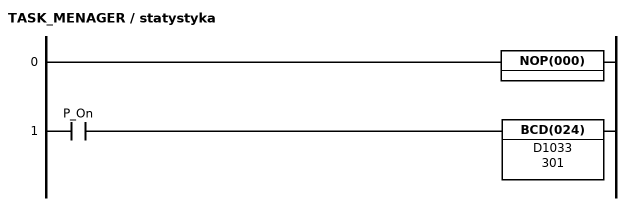
; [picture p24: TASK_MENAGER / statystyka, rungs 0-1]
; rung 0
NOP(000)
; rung 1
LD P_On
BCD(024) D1033 301

### Section wyświetlacz

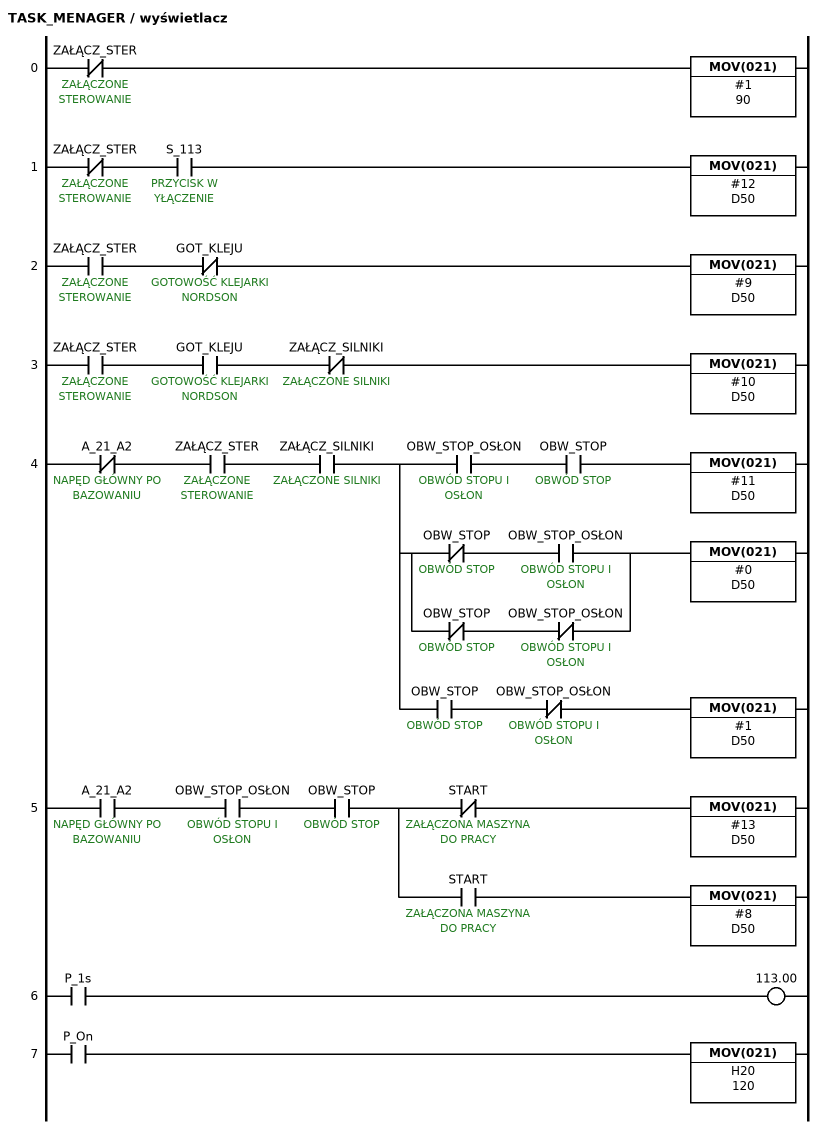
; rung 0
LDNOT ZAŁĄCZ_STER  ; ZAŁĄCZONE STEROWANIE
MOV(021) #1 90
; rung 1
LDNOT ZAŁĄCZ_STER  ; ZAŁĄCZONE STEROWANIE
AND S_113  ; PRZYCISK W YŁĄCZENIE
MOV(021) #12 D50
; rung 2
LD ZAŁĄCZ_STER  ; ZAŁĄCZONE STEROWANIE
ANDNOT GOT_KLEJU  ; GOTOWOŚĆ KLEJARKI NORDSON
MOV(021) #9 D50
; rung 3
LD ZAŁĄCZ_STER  ; ZAŁĄCZONE STEROWANIE
AND GOT_KLEJU  ; GOTOWOŚĆ KLEJARKI NORDSON
ANDNOT ZAŁĄCZ_SILNIKI  ; ZAŁĄCZONE SILNIKI
MOV(021) #10 D50
; rung 4
LDNOT A_21_A2  ; NAPĘD GŁÓWNY PO BAZOWANIU
AND ZAŁĄCZ_STER  ; ZAŁĄCZONE STEROWANIE
AND ZAŁĄCZ_SILNIKI  ; ZAŁĄCZONE SILNIKI
OUT TR0
AND OBW_STOP_OSŁON  ; OBWÓD STOPU I OSŁON
AND OBW_STOP  ; OBWÓD STOP
MOV(021) #11 D50
LD TR0
LDNOT OBW_STOP  ; OBWÓD STOP
AND OBW_STOP_OSŁON  ; OBWÓD STOPU I OSŁON
LDNOT OBW_STOP  ; OBWÓD STOP
ANDNOT OBW_STOP_OSŁON  ; OBWÓD STOPU I OSŁON
ORLD
ANDLD
MOV(021) #0 D50
LD TR0
AND OBW_STOP  ; OBWÓD STOP
ANDNOT OBW_STOP_OSŁON  ; OBWÓD STOPU I OSŁON
MOV(021) #1 D50
; rung 5
LD A_21_A2  ; NAPĘD GŁÓWNY PO BAZOWANIU
AND OBW_STOP_OSŁON  ; OBWÓD STOPU I OSŁON
AND OBW_STOP  ; OBWÓD STOP
OUT TR0
ANDNOT START  ; ZAŁĄCZONA MASZYNA DO PRACY
MOV(021) #13 D50
LD TR0
AND START  ; ZAŁĄCZONA MASZYNA DO PRACY
MOV(021) #8 D50
; rung 6
LD P_1s
OUT 113.00
; rung 7
LD P_On
MOV(021) H20 120
; rung 8
END(001)